// TwinCAT 3 PLC project PLC_VFD
// ProgramVersion: 3.1.4023.0
// libraries:
//   Tc2_Standard, * (Beckhoff Automation GmbH)
//   Tc2_System, * (Beckhoff Automation GmbH)
//   Tc3_Module, * (Beckhoff Automation GmbH)
//   VisuSymbols,3.5.10.0,System
// project tree:
//   DUTs/ ST_Motor_IO.TcDUT, ST_Motor_Params.TcDUT
//   / GlobalTextList.TcGTLO, PlcTask.TcTTO
//   GVLs/ GVL.TcGVL, HMI.TcGVL
//   POUs/ MAIN.TcPOU, FB_Motor.TcPOU
// real-time tasks:
//   TASK PlcTask: cycle T#10ms, priority 20, ADS port 350
// I/O:
//   DEVICE Master (EtherCAT), AmsNetId 172.19.38.34.4.1
//     Drive 1 (FECA-01 v1.31 and ACS880 AINFC v2.62) [FECA-01 v1.31 and ACS880 AINFC v2.62]
// variable links:
//   PLC_VFD/PLC_VFD Instance <-> Master (EtherCAT)/Drive 1 (FECA-01 v1.31 and ACS880 AINFC v2.62)
//     PlcTask Inputs/MAIN.aMotorIO[0].StatusWord <-> TxPDO 21 map/ABB Drives status word
//     PlcTask Inputs/MAIN.aMotorIO[0].iInn_Controller <-> TxPDO 21 map/19.01 Actual operation mode
//     PlcTask Inputs/MAIN.aMotorIO[0].iInn_State <-> InfoData/State
//     PlcTask Inputs/MAIN.aMotorIO[0].rInn_Current <-> TxPDO 21 map/01.07 Motor current
//     PlcTask Inputs/MAIN.aMotorIO[0].rInn_Frequency <-> TxPDO 21 map/01.06 Output frequency
//     PlcTask Inputs/MAIN.aMotorIO[0].rInn_RPM <-> TxPDO 21 map/01.01 Motor speed used
//     PlcTask Inputs/MAIN.aMotorIO[0].rInn_Torque <-> TxPDO 21 map/01.10 Motor torque
//     PlcTask Inputs/MAIN.aMotorIO[0].rInn_Voltage <-> TxPDO 21 map/01.13 Output voltage

CONFIGURATION PLC_VFD
    RESOURCE PLC ON TwinCAT3
        TASK PlcTask(INTERVAL := T#10ms, PRIORITY := 20);
        PROGRAM MAIN WITH PlcTask : MAIN;
    END_RESOURCE
END_CONFIGURATION

// ---- DUTs/ST_Motor_IO.TcDUT
TYPE ST_Motor_IO :
STRUCT
	// Each motor's parameters are read/written through the I/O defined in this struct.
	rInn_RPM			AT%I*	: REAL;
	rInn_Torque			AT%I*	: REAL;
	rInn_Current		AT%I*	: REAL;
	rInn_Voltage		AT%I*	: REAL;
	rInn_Frequency		AT%I*	: REAL;
	iInn_Controller		AT%I*	: UINT;
	iInn_State			AT%I*	: UINT;
	
	rReference			AT%Q*	: REAL;
	iNew_Controller		AT%Q*	: UINT;
	
	StatusWord 			AT%I*	: WORD;
	ControlWord			AT%Q*	: WORD;			
END_STRUCT
END_TYPE

// ---- DUTs/ST_Motor_Params.TcDUT
TYPE ST_Motor_Params :
STRUCT
	// Struct used to update HMI DATAGRID values and ensure selection of editable 
	// HMI DATAGRID array index corresonds to the correct motor object index.
	rRPM				: REAL;
	rTorque				: REAL;
	rCurrent			: REAL;
	rVoltage			: REAL;
	rFrequency			: REAL;
	iControlMethod		: UINT;
	iState				: UINT;
	bSelectMotor		: BOOL;
END_STRUCT
END_TYPE

// ---- GVLs/GVL.TcGVL
{attribute 'qualified_only'}
VAR_GLOBAL
		
	iNumb_Motors			:INT	:= 1;

END_VAR

// ---- GVLs/HMI.TcGVL
{attribute 'qualified_only'}
VAR_GLOBAL
	// Input from HMI
	iReference_Input 			:UINT;
	// Input from HMI
	iControler_Input			:UINT;
	// Input from HMI
	aMotor_Selection 			: ARRAY[0..GVL.iNumb_Motors] OF	BOOL;

END_VAR

// ---- POUs/MAIN.TcPOU
PROGRAM MAIN
VAR
	bFirst_Startup			: BOOL		:= TRUE;
	bEmergencyStop			: BOOL 		:= FALSE;
	
	aMotorList				: ARRAY[0..GVL.iNumb_Motors] OF FB_Motor;
	aMotorParamList			: ARRAY[0..GVL.iNumb_Motors] OF ST_Motor_Params;
	aMotorIO				: ARRAY[0..GVL.iNumb_Motors] OF ST_Motor_IO;			
	
END_VAR

FirstStartup();
EmergencyStop();

MotorParamsUpdater();

METHOD EmergencyStop
VAR_INPUT
END_VAR
VAR
	iCounter	: INT;
END_VAR
	// sets the 2nd bit of each motor objects controlWord to TRUE, wich triggers the drives stop function.
IF bEmergencyStop THEN
	FOR iCounter := 0 TO GVL.iNumb_Motors DO 
		aMotorList[iCounter].ControlWord.2	:= TRUE;	//Emergency stop bit.
	END_FOR
	
END_IF
END_METHOD

METHOD FirstStartup
VAR_INPUT
END_VAR
VAR
	iCounter	:INT;
END_VAR
	// Runs only the at First startup. sets each motor object in arran 10 th and 0 ht bit to TRUE,
	// where the 10th activates the drives remote control mode
	// and the 0th activates the drives READY TO RUN function
	// Also resets EMERGENCY STOP to FALSE.
IF bFirst_Startup THEN
	FOR iCounter := 0 TO GVL.iNumb_Motors DO
		aMotorList[iCounter].ControlWord.10 := TRUE;	// Remote control 
		aMotorList[iCounter].ControlWord.0 := TRUE;		// READY TO RUN
	END_FOR
	bEmergencyStop	:= FALSE;							// Resets EmergencyStop after Restart.
	bFirst_Startup 	:= FALSE;
END_IF
END_METHOD

METHOD MotorParamsUpdater
VAR_INPUT
END_VAR
VAR 
	iCounter: INT;
END_VAR
	// Loop through each motor object in motor array and sets it's parameters acording to reacived values from the drive
	// and updates drive controller and reference if a change is detected from user through the HMI.
FOR iCounter := 0 TO GVL.iNumb_Motors BY 1 DO 
	
		//Updates motor object's parameters according to the drives real time values.
	aMotorList[iCounter].iState_Input 			:= aMotorIO[iCounter].iInn_State;
	aMotorList[iCounter].iController_Input		:= aMotorIO[iCounter].iInn_Controller;
	aMotorList[iCounter].rCurrent_Input			:= aMotorIO[iCounter].rInn_Current;
	aMotorList[iCounter].rReference_Input		:= aMotorIO[iCounter].rInn_Frequency;
	aMotorList[iCounter].rRPM_Input				:= aMotorIO[iCounter].rInn_RPM;
	aMotorList[iCounter].rTorque_Input			:= aMotorIO[iCounter].rInn_Torque;
	aMotorList[iCounter].rVoltage_Input			:= aMotorIO[iCounter].rInn_Voltage;
	
				// Updates Frequency and control method for the current indexed motor
				// in the array, if the corresponding array position in it's Parameter list is TRUE, wich comes from the HMI.
		IF aMotorParamList[iCounter].bSelectMotor = TRUE THEN
			IF (aMotorList[iCounter].iController <> HMI.iControler_Input) THEN
				aMotorList[iCounter].iController_Input	:= HMI.iControler_Input;
				aMotorIO[iCounter].iNew_Controller		:= HMI.iControler_Input;
			END_IF
			IF (aMotorList[iCounter].rReference <> HMI.iReference_Input) THEN
				aMotorList[iCounter].rReference_Input	:= HMI.iReference_Input;
				aMotorIO[iCounter].rReference		:= HMI.iReference_Input;
			END_IF
		END_IF
	
		//  Send motor parameters to an array for display to HMI..
	aMotorParamList[iCounter].iState				:= aMotorList[iCounter].iState;
	aMotorParamList[iCounter].iControlMethod		:= aMotorList[iCounter].iController;
	aMotorParamList[iCounter].rCurrent			:= aMotorList[iCounter].rCurrent;
	aMotorParamList[iCounter].rFrequency			:= aMotorList[iCounter].rReference;
	aMotorParamList[iCounter].rRPM				:= aMotorList[iCounter].rRPM;
	aMotorParamList[iCounter].rTorque			:= aMotorList[iCounter].rTorque;
	aMotorParamList[iCounter].rVoltage			:= aMotorList[iCounter].rVoltage;
		
END_FOR
END_METHOD

END_PROGRAM

// ---- POUs/FB_Motor.TcPOU
FUNCTION_BLOCK FB_Motor
VAR_INPUT
	iState_Input			: UINT;
	iController_Input		: UINT;
	
	rCurrent_Input			: REAL;
	rReference_Input		: REAL;
	rRPM_Input				: REAL;
	rTorque_Input			: REAL;
	rVoltage_Input			: REAL;
	
	StatusWord				: WORD;
	ControlWord				: WORD;
END_VAR
VAR
	iState			: UINT	:= iState_Input;
	iController		: UINT	:= iController_Input;
	
	rCurrent		: REAL	:= rCurrent_Input;
	rReference		: REAL	:= rReference_Input;
	rRPM			: REAL	:= rRPM_Input;
	rTorque			: REAL	:= rTorque_Input;
	rVoltage		: REAL	:= rVoltage_Input;
	
	wControl		: WORD	:= ControlWord;
	wStatus			: WORD	:= StatusWord;
END_VAR

// Designed to hold values Received from the drive and HMI.

END_FUNCTION_BLOCK

// ---- GlobalTextList.TcGTLO
TEXTLIST GlobalTextList
  369 = 'hei'
END_TEXTLIST
